// TwinCAT 3 PLC project PLC
// ProgramVersion: 3.1.0.8
// libraries:
//   Tc2_MC2, * (Beckhoff Automation GmbH)
//   Tc2_Standard, * (Beckhoff Automation GmbH)
//   Tc2_System, * (Beckhoff Automation GmbH)
//   Tc3_Interfaces, * (Beckhoff Automation GmbH)
//   Tc3_Module, * (Beckhoff Automation GmbH)
// project tree:
//   Motion/ AxisCollection.TcPOU, Motion_Parameters.TcGVL
//   Motion/Custom Datatypes/ Motion_Axis.TcDUT (not stored), Motion_AxisGroup.TcDUT (not stored), Motion_FunctionResult.TcDUT (not stored), Motion_HmiToPlc.TcDUT (not stored), Motion_PlcToHmi.TcDUT (not stored)
//   Motion/Version/ Global_Version.TcGVL (not stored)
//   Machine Object/ Machine.TcPOU
//   Tasks/ PlcTask.TcTTO
// real-time tasks:
//   TASK PlcTask: cycle T#10ms, priority 20, ADS port 350
// motion (NC):
//   TASK NC-Task 1 SAF: cycle T#2ms, priority 4, ADS port 501
//   TASK NC-Task 1 SVB: cycle T#10ms, priority 8, ADS port 511
//   AXIS Axis 1 (id 1)
//     OtherSettings: AllowMotionCmdToSlave=true
//     encoder EncType=1
//     drive DrvType=5
//     controller CtrType=1
//       CtrPara: PriorControlFactor=1
//         Observer: BandWidth=20
//   AXIS Axis 2 (id 2)
//     OtherSettings: AllowMotionCmdToSlave=true
//     encoder EncType=1
//     drive DrvType=5
//     controller CtrType=1
//       CtrPara: PriorControlFactor=1
//         Observer: BandWidth=20
//   AXIS Axis 3 (id 3)
//     OtherSettings: AllowMotionCmdToSlave=true
//     encoder EncType=1
//     drive DrvType=5
//     controller CtrType=1
//       CtrPara: PriorControlFactor=1
//         Observer: BandWidth=20
//   AXIS Axis 4 (id 4)
//     OtherSettings: AllowMotionCmdToSlave=true
//     encoder EncType=1
//     drive DrvType=5
//     controller CtrType=1
//       CtrPara: PriorControlFactor=1
//         Observer: BandWidth=20
//   AXIS Axis 5 (id 5)
//     OtherSettings: AllowMotionCmdToSlave=true
//     encoder EncType=1
//     drive DrvType=5
//     controller CtrType=1
//       CtrPara: PriorControlFactor=1
//         Observer: BandWidth=20
//   AXIS Axis 6 (id 6)
//     OtherSettings: AllowMotionCmdToSlave=true
//     encoder EncType=1
//     drive DrvType=5
//     controller CtrType=1
//       CtrPara: PriorControlFactor=1
//         Observer: BandWidth=20
//   AXIS Axis 7 (id 7)
//     OtherSettings: AllowMotionCmdToSlave=true
//     encoder EncType=1
//     drive DrvType=5
//     controller CtrType=1
//       CtrPara: PriorControlFactor=1
//         Observer: BandWidth=20
//   AXIS Axis 8 (id 8)
//     OtherSettings: AllowMotionCmdToSlave=true
//     encoder EncType=1
//     drive DrvType=5
//     controller CtrType=1
//       CtrPara: PriorControlFactor=1
//         Observer: BandWidth=20
//   AXIS Axis 9 (id 9)
//     OtherSettings: AllowMotionCmdToSlave=true
//     encoder EncType=1
//     drive DrvType=5
//     controller CtrType=1
//       CtrPara: PriorControlFactor=1
//         Observer: BandWidth=20
// variable links:
//   PLC/PLC Instance <-> NC-Task 1 SAF/Axes/Axis 1
//     PlcTask Inputs/Machine.AxisGroup[1].AXIS[1].AXIS.NcToPlc <-> Outputs/ToPlc
//     PlcTask Outputs/Machine.AxisGroup[1].AXIS[1].AXIS.PlcToNc <-> Inputs/FromPlc
//   PLC/PLC Instance <-> NC-Task 1 SAF/Axes/Axis 2
//     PlcTask Inputs/Machine.AxisGroup[1].AXIS[2].AXIS.NcToPlc <-> Outputs/ToPlc
//     PlcTask Outputs/Machine.AxisGroup[1].AXIS[2].AXIS.PlcToNc <-> Inputs/FromPlc
//   PLC/PLC Instance <-> NC-Task 1 SAF/Axes/Axis 3
//     PlcTask Inputs/Machine.AxisGroup[1].AXIS[3].AXIS.NcToPlc <-> Outputs/ToPlc
//     PlcTask Outputs/Machine.AxisGroup[1].AXIS[3].AXIS.PlcToNc <-> Inputs/FromPlc
//   PLC/PLC Instance <-> NC-Task 1 SAF/Axes/Axis 4
//     PlcTask Inputs/Machine.AxisGroup[2].AXIS[1].AXIS.NcToPlc <-> Outputs/ToPlc
//     PlcTask Outputs/Machine.AxisGroup[2].AXIS[1].AXIS.PlcToNc <-> Inputs/FromPlc
//   PLC/PLC Instance <-> NC-Task 1 SAF/Axes/Axis 5
//     PlcTask Inputs/Machine.AxisGroup[2].AXIS[2].AXIS.NcToPlc <-> Outputs/ToPlc
//     PlcTask Outputs/Machine.AxisGroup[2].AXIS[2].AXIS.PlcToNc <-> Inputs/FromPlc
//   PLC/PLC Instance <-> NC-Task 1 SAF/Axes/Axis 6
//     PlcTask Inputs/Machine.AxisGroup[2].AXIS[3].AXIS.NcToPlc <-> Outputs/ToPlc
//     PlcTask Outputs/Machine.AxisGroup[2].AXIS[3].AXIS.PlcToNc <-> Inputs/FromPlc
//   PLC/PLC Instance <-> NC-Task 1 SAF/Axes/Axis 7
//     PlcTask Inputs/Machine.AxisGroup[3].AXIS[1].AXIS.NcToPlc <-> Outputs/ToPlc
//     PlcTask Outputs/Machine.AxisGroup[3].AXIS[1].AXIS.PlcToNc <-> Inputs/FromPlc
//   PLC/PLC Instance <-> NC-Task 1 SAF/Axes/Axis 8
//     PlcTask Inputs/Machine.AxisGroup[3].AXIS[2].AXIS.NcToPlc <-> Outputs/ToPlc
//     PlcTask Outputs/Machine.AxisGroup[3].AXIS[2].AXIS.PlcToNc <-> Inputs/FromPlc
//   PLC/PLC Instance <-> NC-Task 1 SAF/Axes/Axis 9
//     PlcTask Inputs/Machine.AxisGroup[3].AXIS[3].AXIS.NcToPlc <-> Outputs/ToPlc
//     PlcTask Outputs/Machine.AxisGroup[3].AXIS[3].AXIS.PlcToNc <-> Inputs/FromPlc

CONFIGURATION PLC
    RESOURCE PLC ON TwinCAT3
        TASK PlcTask(INTERVAL := T#10ms, PRIORITY := 20);
        PROGRAM Machine WITH PlcTask : Machine;
    END_RESOURCE
END_CONFIGURATION

// ---- Motion/Motion_Parameters.TcGVL
VAR_GLOBAL CONSTANT
	MAX_AXES 		: INT := 3;
END_VAR

// ---- Machine Object/Machine.TcPOU
PROGRAM Machine
VAR
	(*Motion Section*)
	AxisGroup : ARRAY[1..3] OF AxisCollection;
	
	(*IO Section*)
	Digital_Sensor			AT %I*		: ARRAY [1..10] OF BOOL;
	HeightThreshold 		AT %I*		: BOOL;
	Cabinet_Open 			AT %I*	  	: BOOL;
	
	(*Machine*)
	Process_Completed					: ARRAY[1..5] OF BOOL;
	Process_Temperature 				: ARRAY[1..5] OF LREAL := [30, 29, 28, 31];
	Process_Quality 					: INT := 90;
	Process_Speed 						: REAL := 30;
	Name								: STRING := 'myMachine';
	Sequence							: INT := 0;
	Sequence_Request					: INT := -1;
	State								: INT := 10;
	State_Request 						: INT := -1;
	
	(*Internal*)
	i,j,k : INT;
	bflag1,bflag2,bflag3,bflag4,bflag5 : BOOL;
END_VAR

CASE State OF
0:	
	IF Sequence_Request > 0 THEN
		Sequence := Sequence_Request;
		Sequence_Request := -1;
	END_IF
	IF State_Request > 0 THEN
		State := State_Request;
		State_Request := -1;
	END_IF
10:
	k := 0;
	FOR i := 1 TO 3 BY 1 DO
		FOR j := 1 TO MAX_AXES BY 1 DO
			IF AxisGroup[i].On(j, TRUE, TRUE, 100) = Motion_FunctionResult.MOTION_OK THEN
				k := k + 1;
				IF k >= MAX_AXES*3 THEN
					State := 0;
				END_IF
			END_IF
		END_FOR
	END_FOR
100:
	CASE Sequence OF
		1 :
			IF NOT bFlag1 THEN 
				IF AxisGroup[1].MoveByDistance(1, 200, 200, 0,0,0) = Motion_FunctionResult.MOTION_OK THEN bFlag1 := TRUE; END_IF
			END_IF
			IF NOT bFlag2 THEN 
				IF AxisGroup[2].MoveByDistance(2, 200, 200, 0,0,0) = Motion_FunctionResult.MOTION_OK THEN bFlag2 := TRUE; END_IF
			END_IF
			IF NOT bFlag3 THEN 
				IF AxisGroup[1].MoveByDistance(3, 200, 200, 0,0,0) = Motion_FunctionResult.MOTION_OK THEN bFlag3 := TRUE; END_IF
			END_IF
			IF bFlag1 AND bFlag2 AND bFlag3 THEN 
				bFlag1 := bFlag2 := bFlag3 := FALSE;
				Sequence := 0;
				State := 0;
			END_IF
	END_CASE
END_CASE




Process_Temperature[1] := Process_Temperature[1] + 0.01;
IF Process_Temperature[1] > 32 THEN
	Process_Temperature[1] := 29.02;
END_IF
Process_Temperature[2] := Process_Temperature[2] + 0.01;
IF Process_Temperature[2] > 32 THEN
	Process_Temperature[2] := 29.12;
END_IF
Process_Temperature[3] := Process_Temperature[3] + 0.01;
IF Process_Temperature[3] > 32 THEN
	Process_Temperature[3] := 30.02;
END_IF
Process_Temperature[4] := Process_Temperature[4] + 0.01;
IF Process_Temperature[4] > 32 THEN
	Process_Temperature[4] := 30.05;
END_IF
Process_Temperature[5] := Process_Temperature[5] + 0.01;
IF Process_Temperature[5] > 32 THEN
	Process_Temperature[5] := 31.01;
END_IF

END_PROGRAM

// ---- Motion/AxisCollection.TcPOU
FUNCTION_BLOCK AxisCollection
VAR_INPUT
END_VAR
VAR_OUTPUT
END_VAR
VAR
	HmiToPlc	: ARRAY[1..MAX_AXES] OF Motion_HmiToPlc;
	PlcToHmi	: ARRAY[1..MAX_AXES] OF Motion_PlcToHmi;
	AXIS		: ARRAY[1..MAX_AXES] OF Motion_Axis;
	fbPower 	: ARRAY [1..MAX_AXES] OF MC_POWER;
	fbReset 	: ARRAY [1..MAX_AXES] OF MC_RESET;
	fbHome		: ARRAY	[1..MAX_AXES] OF MC_HOME;
	fbMoveA 	: ARRAY [1..MAX_AXES] OF MC_MOVEABSOLUTE;
	fbMoveR 	: ARRAY [1..MAX_AXES] OF MC_MOVERELATIVE;
	fbJog		: ARRAY [1..MAX_AXES] OF MC_JOG;
	fbHalt	 	: ARRAY [1..MAX_AXES] OF MC_HALT;
	i			: INT;
	bHmiMode	: BOOL := FALSE;
END_VAR

IF THIS^.HmiMode THEN
	FOR i := 1 TO MAX_AXES BY 1 DO
		ACT_UpdateStatus();
		IF HmiToPlc[i].OFF THEN
			ACT_Off();
		ELSIF HmiToPlc[i].ON THEN 
			ACT_On();
		END_IF
		IF NOT HmiToPlc[i].JOG_MODE THEN 
			Jog_Stop(i);
			IF HmiToPlc[i].HALT THEN 
				ACT_Halt();
			ELSIF HmiToPlc[i].MOVE_ABS THEN
				ACT_MoveToPosition();
			END_IF
			IF HmiToPlc[i].MOVE_REL THEN
				ACT_MoveByDistance();
			END_IF
		ELSE
			ACT_Jog();
		END_IF
	END_FOR
END_IF

METHOD PUBLIC Halt : Motion_FunctionResult
VAR_INPUT
	INDEX : INT;
END_VAR
IF INDEX > MAX_AXES OR INDEX < 1 THEN 
	Halt := Motion_FunctionResult.MOTION_UNKNOWN_AXIS;
ELSE
	fbHalt[INDEX](
		Axis:= AXIS[INDEX].AXIS, 
		Execute:= TRUE );
	fbMoveA[INDEX](
		Axis:= AXIS[INDEX].AXIS, 
		Execute:= FALSE );
	fbMoveR[INDEX](
		Axis:= AXIS[INDEX].AXIS, 
		Execute:= FALSE );
	IF fbHalt[INDEX].Error THEN
		fbHalt[INDEX](
			Axis:= AXIS[INDEX].AXIS, 
			Execute:= FALSE );
		Halt := Motion_FunctionResult.MOTION_ERROR;
	ELSIF fbHalt[INDEX].CommandAborted THEN
		fbHalt[INDEX](
			Axis:= AXIS[INDEX].AXIS, 
			Execute:= FALSE );
		Halt := Motion_FunctionResult.MOTION_COMMAND_ABORTED;
	ELSIF fbHalt[INDEX].Done THEN
		fbHalt[INDEX](
			Axis:= AXIS[INDEX].AXIS, 
			Execute:= FALSE );
		Halt := Motion_FunctionResult.MOTION_OK;
	ELSE
		Halt := Motion_FunctionResult.MOTION_BUSY;
	END_IF
END_IF
END_METHOD

ACTION ACT_Off:
Off(i);
END_ACTION

METHOD PUBLIC MoveToPosition : Motion_FunctionResult
VAR_INPUT
	INDEX 			: INT;
	POSITION		: LREAL;
	VELOCITY		: LREAL;
	ACCELERATION	: LREAL;
	DECELERATION	: LREAL;
	JERK			: LREAL;
END_VAR
IF INDEX > MAX_AXES OR INDEX < 1 AND VELOCITY <= 0 THEN 
	MoveToPosition := Motion_FunctionResult.MOTION_UNKNOWN_AXIS;
ELSE
	fbMoveA[INDEX](
		Axis:= AXIS[INDEX].AXIS, 
		Execute:= TRUE, 
		Position:= POSITION, 
		Velocity:= VELOCITY, 
		Acceleration:= ACCELERATION, 
		Deceleration:= DECELERATION, 
		Jerk:= JERK );
	IF fbMoveA[INDEX].Error THEN
		fbMoveA[INDEX](
			Axis:= AXIS[INDEX].AXIS, 
			Execute:= FALSE );
		MoveToPosition := Motion_FunctionResult.MOTION_ERROR;
	ELSIF fbMoveA[INDEX].CommandAborted THEN
		fbMoveA[INDEX](
			Axis:= AXIS[INDEX].AXIS, 
			Execute:= FALSE );
		MoveToPosition := Motion_FunctionResult.MOTION_COMMAND_ABORTED;
	ELSIF fbMoveA[INDEX].Done THEN
		fbMoveA[INDEX](
			Axis:= AXIS[INDEX].AXIS, 
			Execute:= FALSE );
		MoveToPosition := Motion_FunctionResult.MOTION_OK;
	ELSE
		MoveToPosition := Motion_FunctionResult.MOTION_BUSY;
	END_IF
END_IF
END_METHOD

ACTION ACT_Halt:
CASE Halt(i) OF 
Motion_FunctionResult.MOTION_UNKNOWN_AXIS:
	HmiToPlc[i].HALT := FALSE;
Motion_FunctionResult.MOTION_ERROR:
	HmiToPlc[i].HALT := FALSE;
Motion_FunctionResult.MOTION_OK:
	HmiToPlc[i].HALT := FALSE;
Motion_FunctionResult.MOTION_COMMAND_ABORTED:
	HmiToPlc[i].HALT := FALSE;
Motion_FunctionResult.MOTION_BUSY:
	;
END_CASE
END_ACTION

ACTION ACT_UpdateStatus:
AXIS[i].AXIS.ReadStatus();
PlcToHmi[i].actPos	:= AXIS[i].AXIS.NcToPlc.ActPos;
PlcToHmi[i].actVelo := AXIS[i].AXIS.NcToPlc.ActVelo;
PlcToHmi[i].setPos	:= AXIS[i].AXIS.NcToPlc.SetPos;
PlcToHmi[i].setVelo := AXIS[i].AXIS.NcToPlc.SetVelo;
PlcToHmi[i].controller_override := fbPower[i].Override;
PlcToHmi[i].hasError := AXIS[i].AXIS.Status.Error;
PlcToHmi[i].ErrorID := AXIS[i].AXIS.Status.ErrorID;
PlcToHmi[i].isBwDisabled := NOT fbPower[i].Enable_Negative;
PlcToHmi[i].isFwDisabled := NOT fbPower[i].Enable_Positive;
PlcToHmi[i].isCalibrated := AXIS[i].AXIS.Status.Homed;
PlcToHmi[i].isDisabled := AXIS[i].AXIS.Status.Disabled;
PlcToHmi[i].isInRange := AXIS[i].AXIS.Status.InPositionArea;
PlcToHmi[i].isInTarget := AXIS[i].AXIS.Status.InTargetPosition;
PlcToHmi[i].isNegativeDirection := AXIS[i].AXIS.Status.NegativeDirection;
PlcToHmi[i].isNotMoving := AXIS[i].AXIS.Status.NotMoving;
PlcToHmi[i].isPositiveDirection := AXIS[i].AXIS.Status.PositiveDirection;
END_ACTION

METHOD PUBLIC Off : Motion_FunctionResult
VAR_INPUT
	INDEX : INT;
END_VAR
IF INDEX > MAX_AXES OR INDEX < 1 THEN 
	Off := Motion_FunctionResult.MOTION_UNKNOWN_AXIS;
ELSE
	fbPower[INDEX](
		Axis:= AXIS[INDEX].AXIS, 
		Enable:= FALSE, 
		Enable_Positive:= FALSE, 
		Enable_Negative:= FALSE, 
		Override:= 0 );
	IF fbPower[INDEX].Error THEN
		Off := Motion_FunctionResult.MOTION_ERROR;
	ELSIF NOT fbPower[INDEX].Status THEN
		Off := Motion_FunctionResult.MOTION_OK;
	ELSE
		Off := Motion_FunctionResult.MOTION_BUSY;
	END_IF
END_IF
END_METHOD

METHOD PUBLIC Jog_Start : Motion_FunctionResult
VAR_INPUT
	INDEX		: INT;
	REVERSE		: BOOL := FALSE;
	FAST_MODE	: BOOL := FALSE;
END_VAR
IF FAST_MODE THEN 
	fbJog[INDEX].Mode := MC_JOGMODE_STANDARD_FAST;
ELSE
	fbJog[INDEX].Mode := MC_JOGMODE_STANDARD_SLOW;
END_IF

fbJog[INDEX](
	Axis:= AXIS[INDEX].AXIS, 
	JogForward:= NOT REVERSE, 
	JogBackwards:= REVERSE );
IF fbJog[INDEX].Error THEN 
	Jog_Start := Motion_FunctionResult.MOTION_ERROR;
ELSIF AXIS[INDEX].AXIS.Status.Moving THEN 
	Jog_Start := Motion_FunctionResult.MOTION_OK;
END_IF
END_METHOD

METHOD PUBLIC Jog_Stop : Motion_FunctionResult
VAR_INPUT
	INDEX : INT;
END_VAR
fbJog[INDEX](
	Axis:= AXIS[INDEX].AXIS, 
	JogForward:= FALSE, 
	JogBackwards:= FALSE );
IF fbJog[INDEX].Error THEN 
	Jog_Stop := Motion_FunctionResult.MOTION_ERROR;
ELSE
	Jog_Stop := Motion_FunctionResult.MOTION_OK;
END_IF
END_METHOD

METHOD PUBLIC Home : Motion_FunctionResult
VAR_INPUT
	INDEX : INT;
END_VAR
IF INDEX > MAX_AXES OR INDEX < 1 THEN 
	Home := Motion_FunctionResult.MOTION_UNKNOWN_AXIS;
ELSE
	fbHome[INDEX](
		Axis:= AXIS[INDEX].AXIS, 
		Execute:= TRUE, 
		Position:= 0, 
		HomingMode:= MC_DefaultHoming, 
		bCalibrationCam:= AXIS[INDEX].HOME_CALIBRATION );
	IF fbHome[INDEX].Error THEN
		fbHome[INDEX](
			Axis:= AXIS[INDEX].AXIS, 
			Execute:= FALSE );
		Home := Motion_FunctionResult.MOTION_ERROR;
	ELSIF fbHome[INDEX].CommandAborted THEN
		fbHome[INDEX](
			Axis:= AXIS[INDEX].AXIS, 
			Execute:= FALSE );
		Home := Motion_FunctionResult.MOTION_COMMAND_ABORTED;
	ELSIF fbHome[INDEX].Done THEN
		fbHome[INDEX](
			Axis:= AXIS[INDEX].AXIS, 
			Execute:= FALSE );
		Home := Motion_FunctionResult.MOTION_OK;
	ELSE
		Home := Motion_FunctionResult.MOTION_BUSY;
	END_IF
END_IF
END_METHOD

PROPERTY PUBLIC HmiMode : BOOL
GET
HmiMode := bHmiMode;
END_GET
SET
bHmiMode := HmiMode;
END_SET
END_PROPERTY

ACTION ACT_MoveToPosition:
CASE MoveToPosition(i,HmiToPlc[i].TARGET_POSITION,HmiToPlc[i].TARGET_VELOCITY,HmiToPlc[i].TARGET_ACCELERATION,HmiToPlc[i].TARGET_DECELERATION,HmiToPlc[i].TARGET_JERK) OF
Motion_FunctionResult.MOTION_UNKNOWN_AXIS:
	HmiToPlc[i].MOVE_ABS := FALSE;
Motion_FunctionResult.MOTION_COMMAND_ABORTED: 
	HmiToPlc[i].MOVE_ABS := FALSE;
Motion_FunctionResult.MOTION_ERROR:
	HmiToPlc[i].MOVE_ABS := FALSE;
Motion_FunctionResult.MOTION_BUSY: 
	;
Motion_FunctionResult.MOTION_OK:
	HmiToPlc[i].MOVE_ABS := FALSE;
END_CASE
END_ACTION

METHOD PUBLIC MoveByDistance : Motion_FunctionResult
VAR_INPUT
	INDEX 			: INT;
	DISTANCE 		: LREAL;
	VELOCITY 		: LREAL;
	ACCELERATION 	: LREAL;
	DECELERATION 	: LREAL;
	JERK 			: LREAL;
END_VAR
IF INDEX > MAX_AXES OR INDEX < 1 AND VELOCITY <= 0 THEN 
	MoveByDistance := Motion_FunctionResult.MOTION_UNKNOWN_AXIS;
ELSE
	fbMoveR[INDEX](
		Axis:= AXIS[INDEX].AXIS, 
		Execute:= TRUE, 
		Distance:= DISTANCE, 
		Velocity:= VELOCITY, 
		Acceleration:= ACCELERATION, 
		Deceleration:= DECELERATION, 
		Jerk:= JERK );
	IF fbMoveR[INDEX].Error THEN
		fbMoveR[INDEX](
			Axis:= AXIS[INDEX].AXIS, 
			Execute:= FALSE );
		MoveByDistance := Motion_FunctionResult.MOTION_ERROR;
	ELSIF fbMoveR[INDEX].CommandAborted THEN
		fbMoveR[INDEX](
			Axis:= AXIS[INDEX].AXIS, 
			Execute:= FALSE );
		MoveByDistance := Motion_FunctionResult.MOTION_COMMAND_ABORTED;
	ELSIF fbMoveR[INDEX].Done THEN
		fbMoveR[INDEX](
			Axis:= AXIS[INDEX].AXIS, 
			Execute:= FALSE );
		MoveByDistance := Motion_FunctionResult.MOTION_OK;
	ELSE
		MoveByDistance := Motion_FunctionResult.MOTION_BUSY;
	END_IF
END_IF
END_METHOD

ACTION ACT_MoveByDistance:
CASE MoveByDistance(i,HmiToPlc[i].TARGET_POSITION,HmiToPlc[i].TARGET_VELOCITY,HmiToPlc[i].TARGET_ACCELERATION,HmiToPlc[i].TARGET_DECELERATION,HmiToPlc[i].TARGET_JERK) OF
Motion_FunctionResult.MOTION_UNKNOWN_AXIS:
	HmiToPlc[i].MOVE_REL := FALSE;
Motion_FunctionResult.MOTION_COMMAND_ABORTED: 
	HmiToPlc[i].MOVE_REL := FALSE;
Motion_FunctionResult.MOTION_ERROR:
	HmiToPlc[i].MOVE_REL := FALSE;
Motion_FunctionResult.MOTION_BUSY: 
	;
Motion_FunctionResult.MOTION_OK:
	HmiToPlc[i].MOVE_REL := FALSE;
END_CASE
END_ACTION

ACTION ACT_On:
On(i, HmiToPlc[i].ON_FW, HmiToPlc[i].ON_BW, HmiToPlc[i].CONTROLLER_OVERRIDE);
END_ACTION

ACTION ACT_Reset:
IF Reset(i) = Motion_FunctionResult.MOTION_OK THEN
	HmiToPlc[i].RESET := FALSE;
END_IF
END_ACTION

METHOD On : Motion_FunctionResult
VAR_INPUT
	INDEX : INT;
	ENABLE_FW 	: BOOL;
	ENABLE_BW	: BOOL;
	OVERRIDE	: LREAL;
END_VAR
IF INDEX > MAX_AXES OR INDEX < 1 THEN 
	On := Motion_FunctionResult.MOTION_UNKNOWN_AXIS;
ELSE
	fbPower[INDEX](
		Axis:= AXIS[INDEX].AXIS, 
		Enable:= TRUE, 
		Enable_Positive:= ENABLE_FW, 
		Enable_Negative:= ENABLE_BW, 
		Override:= OVERRIDE );
	IF fbPower[INDEX].Error THEN
		On := Motion_FunctionResult.MOTION_ERROR;
	ELSIF fbPower[INDEX].Status THEN
		On := Motion_FunctionResult.MOTION_OK;
	ELSE
		On := Motion_FunctionResult.MOTION_BUSY;
	END_IF
END_IF
END_METHOD

ACTION ACT_Jog:
IF HmiToPlc[i].JOG_FW_FAST THEN
	Jog_Start(i, FALSE, TRUE);
ELSIF HmiToPlc[i].JOG_FW_SLOW THEN
	Jog_Start(i, FALSE, FALSE);
ELSIF HmiToPlc[i].JOG_BW_FAST THEN
	Jog_Start(i, TRUE, TRUE);
ELSIF HmiToPlc[i].JOG_BW_SLOW THEN
	Jog_Start(i, TRUE, FALSE);
ELSE
	Jog_Stop(i);
END_IF
END_ACTION

PROPERTY PUBLIC AxisCount : INT
GET
AxisCount := MAX_AXES;
END_GET
END_PROPERTY

METHOD PUBLIC Reset : Motion_FunctionResult
VAR_INPUT
	INDEX :INT;
END_VAR
IF INDEX > MAX_AXES OR INDEX < 1 THEN 
	Reset := Motion_FunctionResult.MOTION_UNKNOWN_AXIS;
ELSE
	fbReset[INDEX](
		Axis:= AXIS[INDEX].AXIS, 
		Execute:= TRUE );
	IF fbReset[INDEX].Error THEN
		fbReset[INDEX](
			Axis:= AXIS[INDEX].AXIS, 
			Execute:= FALSE );
		Reset := Motion_FunctionResult.MOTION_ERROR;
	ELSIF fbReset[INDEX].Done THEN
		fbReset[INDEX](
			Axis:= AXIS[INDEX].AXIS, 
			Execute:= FALSE );
		Reset := Motion_FunctionResult.MOTION_OK;
	ELSE
		Reset := Motion_FunctionResult.MOTION_BUSY;
	END_IF
END_IF
END_METHOD

END_FUNCTION_BLOCK
